SUBAPPLICATION Uebung_213b_AUDI (* Standard IEC 61131-3 AUDI_FB_CTU (Adapter Version, UDINT) mit Terminal-Ausgabe *)
  (* Standard: 61131-3; Description: Copyright (c) 2026 Meisterschulen am Ostbahnhof This program and the accompanying materials are made available under the terms of the Eclipse Public License 2.0 which is available at https://www.eclipse.org/legal/epl-2.0/ SPDX-License-Identifier: EPL-2.0 *)
  (* Version 1.1, 2026-04-21, Franz Höpfinger, Meisterschulen am Ostbahnhof, Added terminal output for counter value *)
  (* Version 1.0, 2026-04-21, Franz Höpfinger, Meisterschulen am Ostbahnhof, initial API and implementation (Adapter version) *)
  PACKAGE Uebungen;
  IMPORT Uebungen::const::UT::DefaultPool::OutputNumber_N1;
  IMPORT logiBUS::io::DI::logiBUS_DI::Input_I1;
  IMPORT logiBUS::io::DI::logiBUS_DI::Input_I2;
  IMPORT logiBUS::io::DQ::logiBUS_DO::Output_Q1;
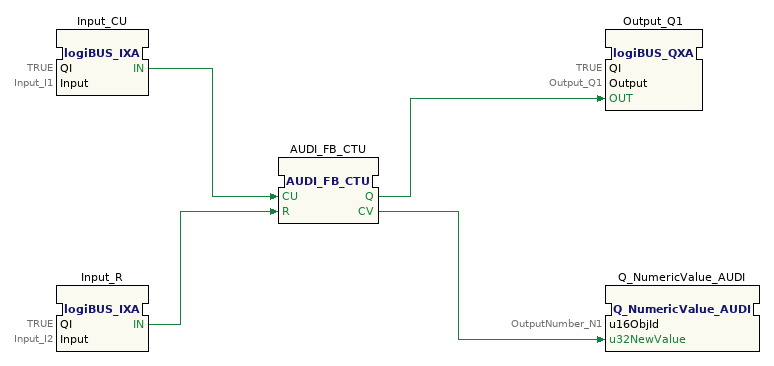
  FBS
    AUDI_FB_CTU : adapter::iec61131::counters::AUDI_FB_CTU;
    Input_CU : logiBUS::io::DI::logiBUS_IXA(QI := TRUE, Input := Input_I1);
    Input_R : logiBUS::io::DI::logiBUS_IXA(QI := TRUE, Input := Input_I2);
    Output_Q1 : logiBUS::io::DQ::logiBUS_QXA(QI := TRUE, Output := Output_Q1);
    Q_NumericValue_AUDI : isobus::UT::Q::Q_NumericValue_AUDI(u16ObjId := OutputNumber_N1);
  END_FBS
  ADAPTER_CONNECTIONS
    Input_CU.IN TO AUDI_FB_CTU.CU;
    Input_R.IN TO AUDI_FB_CTU.R;
    AUDI_FB_CTU.Q TO Output_Q1.OUT;
    AUDI_FB_CTU.CV TO Q_NumericValue_AUDI.u32NewValue;
  END_CONNECTIONS
END_SUBAPPLICATION
